// TIA Portal V19 export
FUNCTION_BLOCK "CabinetDiagReset_10"   // FB13, F_LAD
{ S7_Optimized_Access := 'TRUE' }
   VAR_INPUT
      RESET : Bool;
   END_VAR
BEGIN

REGION Network 1: 1=Acknowledgment for reintegration
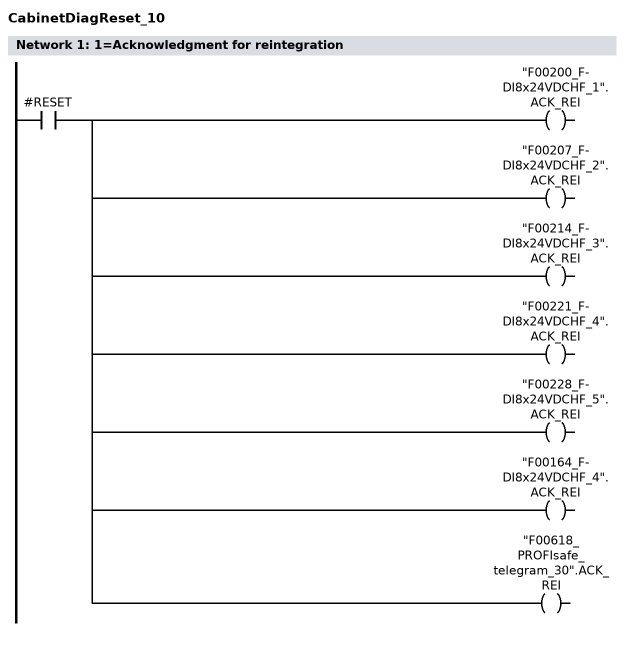
   RUNG wire#powerrail
      Contact( #RESET )
      wire#w1
      Coil( "F00200_F-DI8x24VDCHF_1".ACK_REI )
   END_RUNG
   RUNG wire#w1
      Coil( "F00207_F-DI8x24VDCHF_2".ACK_REI )
   END_RUNG
   RUNG wire#w1
      Coil( "F00214_F-DI8x24VDCHF_3".ACK_REI )
   END_RUNG
   RUNG wire#w1
      Coil( "F00221_F-DI8x24VDCHF_4".ACK_REI )
   END_RUNG
   RUNG wire#w1
      Coil( "F00228_F-DI8x24VDCHF_5".ACK_REI )
   END_RUNG
   RUNG wire#w1
      Coil( "F00164_F-DI8x24VDCHF_4".ACK_REI )
   END_RUNG
   RUNG wire#w1
      Coil( "F00618_PROFIsafe_telegram_30".ACK_REI )
   END_RUNG
   // the same network as SCL:
   "F00200_F-DI8x24VDCHF_1".ACK_REI := #RESET;
   "F00207_F-DI8x24VDCHF_2".ACK_REI := #RESET;
   "F00214_F-DI8x24VDCHF_3".ACK_REI := #RESET;
   "F00221_F-DI8x24VDCHF_4".ACK_REI := #RESET;
   "F00228_F-DI8x24VDCHF_5".ACK_REI := #RESET;
   "F00164_F-DI8x24VDCHF_4".ACK_REI := #RESET;
   "F00618_PROFIsafe_telegram_30".ACK_REI := #RESET;
END_REGION
END_FUNCTION_BLOCK
